# EPICS substitutions: hugo/source/db/Beckhoff_KL/ecmcBK1150.substitutions
file "ecmcBK1X50.template"
{
  pattern {}
          {}
}
